FUNCTION F_AtomicNumberLookup : INT
VAR_INPUT
    sMaterialName : T_MaxString;
END_VAR
VAR
    fbAtomicNumber : FB_AtomicNumber;
END_VAR


fbAtomicNumber(
    sName := sMaterialName
);

IF fbAtomicNumber.bFound THEN
    F_AtomicNumberLookup := fbAtomicNumber.nValue;
ELSE
    F_AtomicNumberLookup := -1;    
END_IF

END_FUNCTION

(* stored: Version 1.1.0.1
   POU F_AtomicNumberLookup: Id {b9771525-53c0-4cfa-a846-c753c62a00cd}, SpecialFunc None *)
